// TIA Portal V21 export
DATA_BLOCK "HmiDB"   // DB4
{ S7_Optimized_Access := 'TRUE' }
// stored: MemoryReserve 100
   VAR
      ksd1 { S7_SetPoint := 'True'} : "coneCrusherHMIs";
      ksd1Sim { S7_SetPoint := 'True'} : "coneCrusherSimHMI";
   END_VAR
BEGIN
   ksd1Sim.cmdWord := 16#1;
   ksd1Sim.ambientTemp := 20.0;
END_DATA_BLOCK
